FUNCTION_BLOCK FB_Normalize_Joystick
VAR_INPUT
	nRawInput : INT;
	fMaxSignal : LREAL;
	fMinSignal : LREAL;
END_VAR
VAR_OUTPUT
	fNormalizedInput : LREAL;
END_VAR
VAR
END_VAR

fNormalizedInput := (INT_TO_LREAL(nRawInput) - 32767.0/2.0) / (32767.0/2.0);

fNormalizedInput := LIMIT(fMinSignal,fNormalizedInput,fMaxSignal);

END_FUNCTION_BLOCK

(* stored: Version 1.1.0.1, ProductVersion 3.1.4024.12
   POU FB_Normalize_Joystick: Id {f566c25e-ef78-4af9-844d-403d72ec68ca}, SpecialFunc None *)
